FUNCTION_BLOCK FB_BufferMetKlep
VAR_INPUT
	i_xAbort		 	: BOOL;
	i_eStartStop 		: eStartStop;
	i_xLightSensor 		: BOOL;
	i_xNextEmpty		: BOOL;
	i_xPreviousEmptying	: BOOL;
	i_xAlarmReset		: BOOL;
	i_eNextState		: eSingleState;
	i_eModus			: eModus := eModus.Auto;
	i_xManualCmdMotor	: BOOL;
END_VAR
VAR_OUTPUT
	o_eState 			: eSingleState := eSinglestate.Idle;
	o_xMotor 			: BOOL := FALSE;
	o_xErrorGeneral 	: BOOL := FALSE;
	o_xAlarmGeneral		: BOOL;
	o_xGivingToNext		: BOOL;
	o_xEmpty			: BOOL	:= TRUE;
	o_sStateString 		: STRING(30);
END_VAR
VAR
	xError					: BOOL;
	tonError	 			: TON;
	fbBlinking 				: FB_Blinking;
	
	fbKlep 					: FB_Klep;
	eValveCurrentPosition	: eValvePosition;
	SIMFUNCTIONING: BOOL :=1;
END_VAR

//-------------------------------------------------------------------------------------------------------------------------
//init objects
fbKlep(	i_eState 						:= o_eState,
		i_eModus						:= i_eModus,
		i_eAutoWantedPosition 			:= (*Set in this FB*),
		i_eManualWantedPosition 		:= (*Used in HMI*),
		i_xHallSensorIn 				:= ,
		i_xHallSensorOut 				:= ,
		i_xWarningReset 				:= (*Used in HMI*),
		i_xAlarmReset 					:= (*Used in HMI*),
		o_eCurrentPosition 				=> eValveCurrentPosition,	
		o_xMagnetValve					=> ,
		o_xWarningPositionDown 			=> (*Used in HMI*),
		o_xErrorPositionUpOrUnknow		=> (*Used in HMI*),
		o_xAlarmPositionUpOrUnknow		=> (*Used in HMI*));

//-------------------------------------------------------------------------------------------------------------------------
//Change the state
//execute
IF NOT (i_eModus = eModus.Off) AND (i_eStartStop = eStartStop.Start) AND NOT i_xAbort AND NOT xError THEN
	o_eState := eSingleState.Execute;
END_IF

//stop request
IF i_eStartStop = eStartStop.Stop THEN
	o_eState := eSingleState.Stopping;
END_IF

//stopping
IF o_eState = eSingleState.Stopping AND o_xMotor = FALSE THEN
	o_eState := eSingleState.Stopped;
END_IF

//suspening
IF (NOT i_xAbort AND NOT (o_eState = eSingleState.Stopped))  AND 
   (i_eNextState = eSingleState.Suspended OR
    i_eNextState = eSingleState.Stopped   OR
    i_eNextState = eSingleState.Aborted) THEN
	o_eState := eSingleState.Suspending;
END_IF

//suspended
IF o_eState = eSingleState.Suspending AND o_xMotor = FALSE THEN
	o_eState := eSingleState.Suspended;
END_IF

IF i_xAbort THEN
	o_eState := eSingleState.Aborting;
END_IF

//aborted
IF o_eState = eSingleState.Aborting AND o_xMotor = FALSE THEN
	o_eState := eSingleState.aborted;
END_IF

//-----------------------------------------------------------------------------------------------------------------------------------------
//Check error and set error, alarm and state = aboarting
tonError(IN := NOT i_xLightSensor AND o_xMotor, PT := T#20S);
IF  o_xMotor AND tonError.Q THEN
    o_eState := eSingleState.Aborting;
	
	IF tonError.Q THEN
		xError := TRUE;
		o_xAlarmGeneral := TRUE;
	END_IF
END_IF;

//blinking error
IF xError THEN
	fbBlinking(io_xBlinking:= o_xErrorGeneral);
ELSIF NOT xError AND o_xAlarmGeneral THEN
	o_xErrorGeneral := TRUE;
ELSE
	o_xErrorGeneral := FALSE;
END_IF;

//----------------------------------------------------------------------------------------------------------------------------------------
//motor on
IF (i_eModus = eModus.Auto) AND 
	(o_eState = eSingleState.Execute AND i_xPreviousEmptying AND NOT i_xLightSensor OR 
	o_eState = eSingleState.Execute AND i_xLightSensor AND i_xNextEmpty AND eValveCurrentPosition = eValvePosition.Down) OR
	(i_eModus = eModus.Manual AND i_xManualCmdMotor) THEN

	o_xMotor := TRUE;
END_IF

//motor off 
IF (i_eModus = eModus.Auto) AND 
	(o_eState = eSingleState.Execute AND i_xLightSensor AND NOT i_xNextEmpty OR 
	o_eState = eSingleState.Stopping OR
	o_eState = eSingleState.Suspending OR
	o_eState = eSingleState.Aborting) OR
	(i_eModus = eModus.Manual AND NOT i_xManualCmdMotor) OR 
	(o_xEmpty AND NOT i_xPreviousEmptying AND NOT (i_eModus = eModus.Manual)) OR
	NOT(eValveCurrentPosition = eValvePosition.Down) THEN

	o_xMotor := FALSE;		
END_IF

//----------------------------------------------------------------------------------------------------------------------------------------
//klep position and write o_xGivingToNext
IF o_eState = eSingleState.Execute AND i_xLightSensor AND NOT i_xNextEmpty THEN
	fbKlep(i_eAutoWantedPosition 		:= eValvePosition.Up);
	o_xGivingToNext := FALSE;
ELSIF o_eState = eSingleState.Execute AND i_xLightSensor AND i_xNextEmpty THEN
	fbKlep(i_eAutoWantedPosition := eValvePosition.Down);
	IF fbKlep.o_eCurrentPosition = eValvePosition.Down THEN
		o_xGivingToNext := TRUE;
	END_IF
ELSIF NOT i_xLightSensor AND NOT i_xNextEmpty THEN //then placed on the next buffer
	o_xGivingToNext := FALSE;
END_IF

//----------------------------------------------------------------------------------------------------------------------------------------
//check if buffer is empty
IF NOT i_xLightSensor THEN
	o_xEmpty := TRUE;
ELSE
	o_xEmpty := FALSE;
END_IF

//-------------------------------------------------------------------------------------------------------------------
//reset alarm and error
IF NOT (o_eState = eSingleState.Aborting) AND i_xLightSensor THEN
	xError := FALSE;
END_IF

//reset alarm
IF i_xAlarmReset AND NOT xError AND NOT (o_eState = eSingleState.Aborting) THEN
	o_xAlarmGeneral := FALSE;
END_IF

//state enum to string for HMI
o_sStateString := F_StateEnumToStringSingleState(o_eState);

//sim
IF gvl.g_xSimulationActive THEN
	IF SIMFUNCTIONING THEN 
		IF i_xPreviousEmptying AND o_xMotor AND gvl.Timerlong.Q AND NOT i_xLightSensor THEN
			i_xLightSensor:=1;
		ELSIF o_xGivingToNext AND o_xMotor AND gvl.Timerlong.Q AND i_xLightSensor THEN
			i_xLightSensor:=0;
		END_IF
	END_IF
END_IF

END_FUNCTION_BLOCK

(* stored: Version 1.1.0.1
   POU FB_BufferMetKlep: Id {f9dd43b7-7628-4dc2-9e96-b2516dfede7d}, SpecialFunc None *)
